(* IEC 61131-3 sources: mect_apps/TP1070_01_C/Monitoring/plc, 9 files *)

(* ---- Crosstable.gvl ---- *)
VAR_GLOBAL
	HeatingEnable AT %QX0.4.0:BOOL;
	HeatingSetPoint_A AT %QW0.8:INT;	(* piano sopra *)
	HeatingSetPoint_B AT %QW0.12:INT;	(* piano terra *)
	HeatingSetPoint_C AT %QW0.16:INT;	(* piano sotto *)
	HeatingDelta AT %QW0.20:INT;
	CoolingEnable AT %QX0.44.0:BOOL;
	CoolingSetPoint_A AT %QW0.48:INT;	(* piano sopra *)
	CoolingSetPoint_B AT %QW0.52:INT;	(* piano terra *)
	CoolingSetPoint_C AT %QW0.56:INT;	(* piano sotto *)
	SavedAlarmStatus AT %QW0.752:UINT;
	SavedAlarmConfig AT %QD0.756:UDINT;
	openvpn_restart_times AT %QD0.768:UDINT;
	is_PPP0_ON AT %QX0.772.0:BOOL;	(* isUP_ppp0() *)
	is_TUN0_ON AT %QX0.776.0:BOOL;	(* isUP_tun0() *)
	is_Caldaia_ON AT %QX0.780.0:BOOL;
	XX_Baudrate AT %IW0.804:UINT;	(* Baudrate MPNC005 device *)
	XX_NodeID AT %IW0.808:UINT;	(* Address MPNC005 device *)
	XX_HeartBeat AT %ID0.812:UDINT;	(* Life time MPNC005 device *)
	XX_AnInConf_A AT %QW0.816:UINT;	(* Analog inputs configuration MPNC030 module A *)
	XX_AnInConf_B AT %QW0.820:UINT;	(* Analog inputs configuration MPNC030 module B *)
	XX_AnInConf_C AT %QW0.824:UINT;	(* Analog inputs configuration MPNC030 module C *)
	XX_AnIn_A_1 AT %IW0.832:INT;	(* Analog input 1 value MPNC030 module A *)
	XX_AnIn_A_2 AT %IW0.836:INT;	(* Analog input 2 value MPNC030 module A *)
	XX_AnIn_A_3 AT %IW0.840:INT;	(* Analog input 3 value MPNC030 module A *)
	XX_AnIn_A_4 AT %IW0.844:INT;	(* Analog input 4 value MPNC030 module A *)
	XX_AnIn_B_1 AT %IW0.848:INT;	(* Analog input 1 value MPNC030 module B *)
	XX_AnIn_B_2 AT %IW0.852:INT;	(* Analog input 2 value MPNC030 module B *)
	XX_AnIn_B_3 AT %IW0.856:INT;	(* Analog input 3 value MPNC030 module B *)
	XX_AnIn_B_4 AT %IW0.860:INT;	(* Analog input 4 value MPNC030 module B *)
	XX_AnIn_C_1 AT %IW0.864:INT;	(* Analog input 1 value MPNC030 module C *)
	XX_AnIn_C_2 AT %IW0.868:INT;	(* Analog input 2 value MPNC030 module C *)
	XX_AnIn_C_3 AT %IW0.872:INT;	(* Analog input 3 value MPNC030 module C *)
	XX_AnIn_C_4 AT %IW0.876:INT;	(* Analog input 4 value MPNC030 module C *)
	XX_DigOut_A_1 AT %QX0.896.0:BOOL;	(* Digital output value bit 1 MPNC020 02 module A *)
	XX_DigOut_A_2 AT %QX0.900.0:BOOL;	(* Digital output value bit 2 MPNC020 02 module A *)
	XX_DigOut_A_3 AT %QX0.904.0:BOOL;	(* Digital output value bit 3 MPNC020 02 module A *)
	XX_DigOut_A_4 AT %QX0.908.0:BOOL;	(* Digital output value bit 4 MPNC020 02 module A *)
	XX_DigOut_A_5 AT %QX0.912.0:BOOL;	(* Digital output value bit 5 MPNC020 02 module A *)
	XX_DigOut_A_6 AT %QX0.916.0:BOOL;	(* Digital output value bit 6 MPNC020 02 module A *)
	XX_DigOut_A_7 AT %QX0.920.0:BOOL;	(* Digital output value bit 7 MPNC020 02 module A *)
	XX_DigOut_A_8 AT %QX0.924.0:BOOL;	(* Digital output value bit 8 MPNC020 02 module A *)
	XX_DigOut_A_9 AT %QX0.928.0:BOOL;	(* Digital output value bit 9 MPNC020 02 module A *)
	XX_DigOut_A_10 AT %QX0.932.0:BOOL;	(* Digital output value bit 10 MPNC020 02 module A *)
	XX_DigOut_A_11 AT %QX0.936.0:BOOL;	(* Digital output value bit 11 MPNC020 02 module A *)
	XX_DigOut_A_12 AT %QX0.940.0:BOOL;	(* Digital output value bit 12 MPNC020 02 module A *)
	XX_DigOut_A_13 AT %QX0.944.0:BOOL;	(* Digital output value bit 13 MPNC020 02 module A *)
	XX_DigOut_A_14 AT %QX0.948.0:BOOL;	(* Digital output value bit 14 MPNC020 02 module A *)
	XX_DigOut_A_15 AT %QX0.952.0:BOOL;	(* Digital output value bit 15 MPNC020 02 module A *)
	XX_DigOut_A_16 AT %QX0.956.0:BOOL;	(* Digital output value bit 16 MPNC020 02 module A *)
	XX_DigIn_A_1 AT %IX0.1152.0:BOOL;	(* Digital input value bit 1 MPNC020 01 module A *)
	XX_DigIn_A_2 AT %IX0.1156.0:BOOL;	(* Digital input value bit 2 MPNC020 01 module A *)
	XX_DigIn_A_3 AT %IX0.1160.0:BOOL;	(* Digital input value bit 3 MPNC020 01 module A *)
	XX_DigIn_A_4 AT %IX0.1164.0:BOOL;	(* Digital input value bit 4 MPNC020 01 module A *)
	XX_DigIn_A_5 AT %IX0.1168.0:BOOL;	(* Digital input value bit 5 MPNC020 01 module A *)
	XX_DigIn_A_6 AT %IX0.1172.0:BOOL;	(* Digital input value bit 6 MPNC020 01 module A *)
	XX_DigIn_A_7 AT %IX0.1176.0:BOOL;	(* Digital input value bit 7 MPNC020 01 module A *)
	XX_DigIn_A_8 AT %IX0.1180.0:BOOL;	(* Digital input value bit 8 MPNC020 01 module A *)
	XX_DigIn_A_9 AT %IX0.1184.0:BOOL;	(* Digital input value bit 9 MPNC020 01 module A *)
	XX_DigIn_A_10 AT %IX0.1188.0:BOOL;	(* Digital input value bit 10 MPNC020 01 module A *)
	XX_DigIn_A_11 AT %IX0.1192.0:BOOL;	(* Digital input value bit 11 MPNC020 01 module A *)
	XX_DigIn_A_12 AT %IX0.1196.0:BOOL;	(* Digital input value bit 12 MPNC020 01 module A *)
	XX_DigIn_A_13 AT %IX0.1200.0:BOOL;	(* Digital input value bit 13 MPNC020 01 module A *)
	XX_DigIn_A_14 AT %IX0.1204.0:BOOL;	(* Digital input value bit 14 MPNC020 01 module A *)
	XX_DigIn_A_15 AT %IX0.1208.0:BOOL;	(* Digital input value bit 15 MPNC020 01 module A *)
	XX_DigIn_A_16 AT %IX0.1212.0:BOOL;	(* Digital input value bit 16 MPNC020 01 module A *)
	XX_DigIn_B_1 AT %IX0.1216.0:BOOL;	(* Digital input value bit 1 MPNC020 01 module B *)
	XX_DigIn_B_2 AT %IX0.1220.0:BOOL;	(* Digital input value bit 2 MPNC020 01 module B *)
	XX_DigIn_B_3 AT %IX0.1224.0:BOOL;	(* Digital input value bit 3 MPNC020 01 module B *)
	XX_DigIn_B_4 AT %IX0.1228.0:BOOL;	(* Digital input value bit 4 MPNC020 01 module B *)
	XX_DigIn_B_5 AT %IX0.1232.0:BOOL;	(* Digital input value bit 5 MPNC020 01 module B *)
	XX_DigIn_B_6 AT %IX0.1236.0:BOOL;	(* Digital input value bit 6 MPNC020 01 module B *)
	XX_DigIn_B_7 AT %IX0.1240.0:BOOL;	(* Digital input value bit 7 MPNC020 01 module B *)
	XX_DigIn_B_8 AT %IX0.1244.0:BOOL;	(* Digital input value bit 8 MPNC020 01 module B *)
	XX_DigIn_B_9 AT %IX0.1248.0:BOOL;	(* Digital input value bit 9 MPNC020 01 module B *)
	XX_DigIn_B_10 AT %IX0.1252.0:BOOL;	(* Digital input value bit 10 MPNC020 01 module B *)
	XX_DigIn_B_11 AT %IX0.1256.0:BOOL;	(* Digital input value bit 11 MPNC020 01 module B *)
	XX_DigIn_B_12 AT %IX0.1260.0:BOOL;	(* Digital input value bit 12 MPNC020 01 module B *)
	XX_DigIn_B_13 AT %IX0.1264.0:BOOL;	(* Digital input value bit 13 MPNC020 01 module B *)
	XX_DigIn_B_14 AT %IX0.1268.0:BOOL;	(* Digital input value bit 14 MPNC020 01 module B *)
	XX_DigIn_B_15 AT %IX0.1272.0:BOOL;	(* Digital input value bit 15 MPNC020 01 module B *)
	XX_DigIn_B_16 AT %IX0.1276.0:BOOL;	(* Digital input value bit 16 MPNC020 01 module B *)
	XX_Reserved_1 AT %IW0.1408:UINT;
	XX_Reserved_2 AT %IW0.1412:UINT;
	XX_ColdJunctionT AT %IW0.1416:INT;	(* Cold junction temperature value *)
	XX_Reserved_3 AT %IW0.1420:UINT;
	XX_Reserved_4 AT %IW0.1424:UINT;
	XX_Reboot AT %QW0.1428:INT;	(* MPNC006 chain reboot *)
	XX_ModulesNumber AT %IW0.1432:UINT;	(* Number of modules *)
	XX_AnInConf_1 AT %QW0.1436:UINT;	(* Analog input 1 configuration MPNC005 *)
	XX_AnInConf_2 AT %QW0.1440:UINT;	(* Analog input 2 configuration MPNC005 *)
	XX_AnIn_1 AT %IW0.1444:INT;	(* Analog input 1 value MPNC005 *)
	XX_AnIn_2 AT %IW0.1448:INT;	(* Analog input 2 value MPNC005 *)
	XX_DigDir_1 AT %QX0.1452.0:BOOL;	(* Digital IO 1 configuration MPNC005 *)
	XX_DigDir_2 AT %QX0.1456.0:BOOL;	(* Digital IO 2 configuration MPNC005 *)
	XX_DigDir_3 AT %QX0.1460.0:BOOL;	(* Digital IO 3 configuration MPNC005 *)
	XX_DigDir_4 AT %QX0.1464.0:BOOL;	(* Digital IO 4 configuration MPNC005 *)
	XX_DigDir_5 AT %QX0.1468.0:BOOL;	(* Digital IO 5 configuration MPNC005 *)
	XX_DigDir_6 AT %QX0.1472.0:BOOL;	(* Digital IO 6 configuration MPNC005 *)
	XX_DigDir_7 AT %QX0.1476.0:BOOL;	(* Digital IO 7 configuration MPNC005 *)
	XX_DigDir_8 AT %QX0.1480.0:BOOL;	(* Digital IO 8 configuration MPNC005 *)
	XX_DigIn_1 AT %IX0.1484.0:BOOL;	(* Digital input 1 value MPNC005 *)
	XX_DigIn_2 AT %IX0.1488.0:BOOL;	(* Digital input 2 value MPNC005 *)
	XX_DigIn_3 AT %IX0.1492.0:BOOL;	(* Digital input 3 value MPNC005 *)
	XX_DigIn_4 AT %IX0.1496.0:BOOL;	(* Digital input 4 value MPNC005 *)
	XX_DigIn_5 AT %IX0.1500.0:BOOL;	(* Digital input 5 value MPNC005 *)
	XX_DigIn_6 AT %IX0.1504.0:BOOL;	(* Digital input 6 value MPNC005 *)
	XX_DigIn_7 AT %IX0.1508.0:BOOL;	(* Digital input 7 value MPNC005 *)
	XX_DigIn_8 AT %IX0.1512.0:BOOL;	(* Digital input 8 value MPNC005 *)
	XX_DigOut_1 AT %QX0.1516.0:BOOL;	(* Digital output 1 value MPNC005 *)
	XX_DigOut_2 AT %QX0.1520.0:BOOL;	(* Digital output 2 value MPNC005 *)
	XX_DigOut_3 AT %QX0.1524.0:BOOL;	(* Digital output 3 value MPNC005 *)
	XX_DigOut_4 AT %QX0.1528.0:BOOL;	(* Digital output 4 value MPNC005 *)
	XX_DigOut_5 AT %QX0.1532.0:BOOL;	(* Digital output 5 value MPNC005 *)
	XX_DigOut_6 AT %QX0.1536.0:BOOL;	(* Digital output 6 value MPNC005 *)
	XX_DigOut_7 AT %QX0.1540.0:BOOL;	(* Digital output 7 value MPNC005 *)
	XX_DigOut_8 AT %QX0.1544.0:BOOL;	(* Digital output 8 value MPNC005 *)
	XX_AnInFltr_1 AT %QW0.1548:UINT;	(* Analog input filter 1 MPNC006 *)
	XX_AnInFltr_2 AT %QW0.1552:UINT;	(* Analog input filter 2 MPNC006 *)
	XX_WatchDog AT %QW0.1556:UINT;	(* WatchDog Timer in Seconds *)
	XX_FirmwareVer AT %IW0.1644:UINT;	(* Firmware release MPNC006 *)
	XX_StatusWord AT %IW0.1648:UINT;	(* Status word MPNC006 *)
	SystemVoltage_0 AT %ID0.1656:REAL;	(* 0x0A 0x100C Tensione in V (PRINCIPALE) *)
	SysPowerFactor_0 AT %ID0.1660:REAL;	(* 0x0A 0x101E Fattore di Potenza 0 (PRINCIPALE) *)
	SysActivePower_0 AT %ID0.1664:REAL;	(* 0x0A 0x1026 Potenza Attiva 0 in W (PRINCIPALE) *)
	SysImpActiveEnergy_0 AT %ID0.1668:REAL;	(* 0x0A 0x1106 Energia Attiva Importata 0 in Wh (PRINCIPALE) *)
	SysExpActiveEnergy_0 AT %ID0.1672:REAL;	(* 0x0A 0x110E Energia Attiva Esportata 0 in Wh (PRINCIPALE) *)
	SysActivePower_1 AT %ID0.1676:REAL;	(* 0x0B 0x1026 Potenza Attiva 0 in W (FOTOVOLTAICO) *)
	SysImpActiveEnergy_1 AT %ID0.1680:REAL;	(* 0x0B 0x1106 Energia Attiva Importata 1 in Wh (FOTOVOLTAICO) *)
	SysExpActiveEnergy_1 AT %ID0.1684:REAL;	(* 0x0B 0x110E Energia Attiva Esportata 0 in Wh (FOTOVOLTAICO) *)
	SysActivePower_2 AT %ID0.1688:REAL;	(* 0x0C 0x1026 Potenza Attiva 0 in W (ESTERNI) *)
	SysImpActiveEnergy_2 AT %ID0.1692:REAL;	(* 0x0C 0x1106 Energia Attiva Importata 0 in Wh (ESTERNI) *)
	SysActivePower_3 AT %ID0.1696:REAL;	(* 0x0D 0x1026 Potenza Attiva 0 in W (PIANO SOPRA) *)
	SysImpActiveEnergy_3 AT %ID0.1700:REAL;	(* 0x0D 0x1106 Energia Attiva Importata 0 in Wh (PIANO SOPRA) *)
	SysActivePower_4 AT %ID0.1704:REAL;	(* 0x0E 0x1026 Potenza Attiva 0 in W (PIANO TERRA) *)
	SysImpActiveEnergy_4 AT %ID0.1708:REAL;	(* 0x0E 0x1106 Energia Attiva Importata 0 in Wh (PIANO TERRA) *)
	SysActivePower_5 AT %ID0.1712:REAL;	(* 0x0F 0x1026 Potenza Attiva 0 in W (PIANO SOTTO) *)
	SysImpActiveEnergy_5 AT %ID0.1716:REAL;	(* 0x0F 0x1106 Energia Attiva Importata 0 in Wh (PIANO SOTTO) *)
	SysActivePower_6 AT %ID0.1720:REAL;	(* 0x10 0x1026 Potenza Attiva 0 in W (AUTO ELETTRICA) *)
	SysImpActiveEnergy_6 AT %ID0.1724:REAL;	(* 0x10 0x1106 Energia Attiva Importata 0 in Wh (AUTO ELETTRICA) *)
	SysActivePower_7 AT %ID0.1728:REAL;	(* 0x11 0x1026 Potenza Attiva 0 in W (DEUMIDIFICATORE) *)
	SysImpActiveEnergy_7 AT %ID0.1732:REAL;	(* 0x11 0x1106 Energia Attiva Importata 0 in Wh (DEUMIDIFICATORE) *)
	SysActivePower_8 AT %ID0.1736:REAL;	(* 0x12 0x1026 Potenza Attiva 0 in W (LAVANDERIA) *)
	SysImpActiveEnergy_8 AT %ID0.1740:REAL;	(* 0x12 0x1106 Energia Attiva Importata 0 in Wh (LAVANDERIA) *)
	SysActivePower_9 AT %ID0.1744:REAL;	(* 0x13 0x1026 Potenza Attiva 0 in W (UPS) *)
	SysApparentPower_9 AT %ID0.1748:REAL;	(* 0x13 0x102E Potenza Apparente 0 in VA (UPS) *)
	SysImpActiveEnergy_9 AT %ID0.1752:REAL;	(* 0x13 0x1106 Energia Attiva Importata 0 in Wh (UPS) *)
	SysActivePower_10 AT %ID0.1756:REAL;	(* 0x14 0x1026 Potenza Attiva 0 in W (Puffer) *)
	SysImpActiveEnergy_10 AT %ID0.1760:REAL;	(* 0x14 0x1106 Energia Attiva Importata 0 in Wh (Puffer) *)
	SysActivePower_11 AT %QD0.1764:REAL;	(* 0x14 0x1026 Potenza Attiva 0 in W (Caldaia) *)
	SysImpActiveEnergy_11 AT %QD0.1768:REAL;	(* 0x14 0x1106 Energia Attiva Importata 0 in Wh (Caldaia) *)
	AlarmStatus AT %QW0.1996:UINT;
	Alarm AT %QX0.2000.0:BOOL;
	OK_DigIn_A_1 AT %QX0.2004.0:BOOL;
	OK_DigIn_A_2 AT %QX0.2008.0:BOOL;
	OK_DigIn_A_3 AT %QX0.2012.0:BOOL;
	OK_DigIn_A_4 AT %QX0.2016.0:BOOL;
	OK_DigIn_A_5 AT %QX0.2020.0:BOOL;
	OK_DigIn_A_6 AT %QX0.2024.0:BOOL;
	OK_DigIn_A_7 AT %QX0.2028.0:BOOL;
	OK_DigIn_A_8 AT %QX0.2032.0:BOOL;
	OK_DigIn_A_9 AT %QX0.2036.0:BOOL;
	OK_DigIn_A_10 AT %QX0.2040.0:BOOL;
	OK_DigIn_A_11 AT %QX0.2044.0:BOOL;
	OK_DigIn_A_12 AT %QX0.2048.0:BOOL;
	OK_DigIn_A_13 AT %QX0.2052.0:BOOL;
	OK_DigIn_A_14 AT %QX0.2056.0:BOOL;
	OK_DigIn_A_15 AT %QX0.2060.0:BOOL;
	OK_DigIn_A_16 AT %QX0.2064.0:BOOL;
	OK_DigIn_B_1 AT %QX0.2068.0:BOOL;
	OK_DigIn_B_2 AT %QX0.2072.0:BOOL;
	OK_DigIn_B_3 AT %QX0.2076.0:BOOL;
	OK_DigIn_B_4 AT %QX0.2080.0:BOOL;
	OK_DigIn_B_5 AT %QX0.2084.0:BOOL;
	OK_DigIn_B_6 AT %QX0.2088.0:BOOL;
	OK_DigIn_B_7 AT %QX0.2092.0:BOOL;
	OK_DigIn_B_8 AT %QX0.2096.0:BOOL;
	OK_DigIn_B_9 AT %QX0.2100.0:BOOL;
	OK_DigIn_B_10 AT %QX0.2104.0:BOOL;
	OK_DigIn_B_11 AT %QX0.2108.0:BOOL;
	OK_DigIn_B_12 AT %QX0.2112.0:BOOL;
	OK_DigIn_B_13 AT %QX0.2116.0:BOOL;
	OK_DigIn_B_14 AT %QX0.2120.0:BOOL;
	OK_DigIn_B_15 AT %QX0.2124.0:BOOL;
	OK_DigIn_B_16 AT %QX0.2128.0:BOOL;
	AlarmRising AT %IX0.2132.0:BOOL;
	AlarmArmed_A_1 AT %QX0.2404.0:BOOL;
	AlarmArmed_A_2 AT %QX0.2408.0:BOOL;
	AlarmArmed_A_3 AT %QX0.2412.0:BOOL;
	AlarmArmed_A_4 AT %QX0.2416.0:BOOL;
	AlarmArmed_A_5 AT %QX0.2420.0:BOOL;
	AlarmArmed_A_6 AT %QX0.2424.0:BOOL;
	AlarmArmed_A_7 AT %QX0.2428.0:BOOL;
	AlarmArmed_A_8 AT %QX0.2432.0:BOOL;
	AlarmArmed_A_9 AT %QX0.2436.0:BOOL;
	AlarmArmed_A_10 AT %QX0.2440.0:BOOL;
	AlarmArmed_A_11 AT %QX0.2444.0:BOOL;
	AlarmArmed_A_12 AT %QX0.2448.0:BOOL;
	AlarmArmed_A_13 AT %QX0.2452.0:BOOL;
	AlarmArmed_A_14 AT %QX0.2456.0:BOOL;
	AlarmArmed_A_15 AT %QX0.2460.0:BOOL;
	AlarmArmed_A_16 AT %QX0.2464.0:BOOL;
	AlarmArmed_B_1 AT %QX0.2468.0:BOOL;
	AlarmArmed_B_2 AT %QX0.2472.0:BOOL;
	AlarmArmed_B_3 AT %QX0.2476.0:BOOL;
	AlarmArmed_B_4 AT %QX0.2480.0:BOOL;
	AlarmArmed_B_5 AT %QX0.2484.0:BOOL;
	AlarmArmed_B_6 AT %QX0.2488.0:BOOL;
	AlarmArmed_B_7 AT %QX0.2492.0:BOOL;
	AlarmArmed_B_8 AT %QX0.2496.0:BOOL;
	AlarmArmed_B_9 AT %QX0.2500.0:BOOL;
	AlarmArmed_B_10 AT %QX0.2504.0:BOOL;
	AlarmArmed_B_11 AT %QX0.2508.0:BOOL;
	AlarmArmed_B_12 AT %QX0.2512.0:BOOL;
	AlarmArmed_B_13 AT %QX0.2516.0:BOOL;
	AlarmArmed_B_14 AT %QX0.2520.0:BOOL;
	AlarmArmed_B_15 AT %QX0.2524.0:BOOL;
	AlarmArmed_B_16 AT %QX0.2528.0:BOOL;
	TCP_is_Caldaia_ON AT %QX0.4000.0:BOOL;
	TCP_HeatingEnable AT %QX0.4004.0:BOOL;
	TCP_AnIn_A_1 AT %QW0.4008:INT;	(* Analog input 1 value MPNC030 module A *)
	TCP_AnIn_A_2 AT %QW0.4012:INT;	(* Analog input 2 value MPNC030 module A *)
	TCP_AnIn_A_3 AT %QW0.4016:INT;	(* Analog input 3 value MPNC030 module A *)
	TCP_AnIn_A_4 AT %QW0.4020:INT;	(* Analog input 4 value MPNC030 module A *)
	TCP_AnIn_B_1 AT %QW0.4024:INT;	(* Analog input 1 value MPNC030 module B *)
	TCP_AnIn_B_2 AT %QW0.4028:INT;	(* Analog input 2 value MPNC030 module B *)
	TCP_AnIn_B_3 AT %QW0.4032:INT;	(* Analog input 3 value MPNC030 module B *)
	TCP_AnIn_B_4 AT %QW0.4036:INT;	(* Analog input 4 value MPNC030 module B *)
	TCP_AnIn_C_1 AT %QW0.4040:INT;	(* Analog input 1 value MPNC030 module C *)
	TCP_AnIn_C_2 AT %QW0.4044:INT;	(* Analog input 2 value MPNC030 module C *)
	TCP_AnIn_C_3 AT %QW0.4048:INT;	(* Analog input 3 value MPNC030 module C *)
	TCP_AnIn_C_4 AT %QW0.4052:INT;	(* Analog input 3 value MPNC030 module C *)
	TCP_AnIn_1 AT %QW0.4056:INT;	(* Analog input 1 value MPNC005 *)
	TCP_AnIn_2 AT %QW0.4060:INT;	(* Analog input 2 value MPNC005 *)
	TCP_DigIn_1 AT %QX0.4064.0:BOOL;	(* Digital input 1 value MPNC005 *)
	TCP_DigIn_2 AT %QX0.4068.0:BOOL;	(* Digital input 2 value MPNC005 *)
	TCP_DigIn_3 AT %QX0.4072.0:BOOL;	(* Digital input 3 value MPNC005 *)
	TCP_DigIn_4 AT %QX0.4076.0:BOOL;	(* Digital input 4 value MPNC005 *)
	TCP_DigIn_5 AT %QX0.4080.0:BOOL;	(* Digital input 5 value MPNC005 *)
	TCP_DigIn_6 AT %QX0.4084.0:BOOL;	(* Digital input 6 value MPNC005 *)
	TCP_DigIn_7 AT %QX0.4088.0:BOOL;	(* Digital input 7 value MPNC005 *)
	TCP_DigIn_8 AT %QX0.4092.0:BOOL;	(* Digital input 8 value MPNC005 *)
	TCP_DigOut_1 AT %QX0.4096.0:BOOL;	(* Digital output 1 value MPNC005 *)
	TCP_DigOut_2 AT %QX0.4100.0:BOOL;	(* Digital output 2 value MPNC005 *)
	TCP_DigOut_3 AT %QX0.4104.0:BOOL;	(* Digital output 3 value MPNC005 *)
	TCP_DigOut_4 AT %QX0.4108.0:BOOL;	(* Digital output 4 value MPNC005 *)
	TCP_DigOut_5 AT %QX0.4112.0:BOOL;	(* Digital output 5 value MPNC005 *)
	TCP_DigOut_6 AT %QX0.4116.0:BOOL;	(* Digital output 6 value MPNC005 *)
	TCP_DigOut_7 AT %QX0.4120.0:BOOL;	(* Digital output 7 value MPNC005 *)
	TCP_DigOut_8 AT %QX0.4124.0:BOOL;	(* Digital output 8 value MPNC005 *)
	TCP_SystemVoltage_0 AT %QD0.4132:REAL;	(* 0x0A 0x100C Tensione in V (PRINCIPALE) *)
	TCP_SysPowerFactor_0 AT %QD0.4136:REAL;	(* 0x0A 0x101E Fattore di Potenza 0 (PRINCIPALE) *)
	TCP_SysActivePower_0 AT %QD0.4140:REAL;	(* 0x0A 0x1026 Potenza Attiva 0 in W (PRINCIPALE) *)
	TCP_SysImpActiveEnergy_0 AT %QD0.4144:REAL;	(* 0x0A 0x1106 Energia Attiva Importata 0 in Wh (PRINCIPALE) *)
	TCP_SysExpActiveEnergy_0 AT %QD0.4148:REAL;	(* 0x0A 0x110E Energia Attiva Esportata 0 in Wh (PRINCIPALE) *)
	TCP_SysActivePower_1 AT %QD0.4152:REAL;	(* 0x0B 0x1026 Potenza Attiva 0 in W (FOTOVOLTAICO) *)
	TCP_SysImpActiveEnergy_1 AT %QD0.4156:REAL;	(* 0x0B 0x1106 Energia Attiva Importata 1 in Wh (FOTOVOLTAICO) *)
	TCP_SysExpActiveEnergy_1 AT %QD0.4160:REAL;	(* 0x0B 0x110E Energia Attiva Esportata 0 in Wh (FOTOVOLTAICO) *)
	TCP_SysActivePower_2 AT %QD0.4164:REAL;	(* 0x0C 0x1026 Potenza Attiva 0 in W (ESTERNI) *)
	TCP_SysImpActiveEnergy_2 AT %QD0.4168:REAL;	(* 0x0C 0x1106 Energia Attiva Importata 0 in Wh (ESTERNI) *)
	TCP_SysActivePower_3 AT %QD0.4172:REAL;	(* 0x0D 0x1026 Potenza Attiva 0 in W (PIANO SOPRA) *)
	TCP_SysImpActiveEnergy_3 AT %QD0.4176:REAL;	(* 0x0D 0x1106 Energia Attiva Importata 0 in Wh (PIANO SOPRA) *)
	TCP_SysActivePower_4 AT %QD0.4180:REAL;	(* 0x0E 0x1026 Potenza Attiva 0 in W (PIANO TERRA) *)
	TCP_SysImpActiveEnergy_4 AT %QD0.4184:REAL;	(* 0x0E 0x1106 Energia Attiva Importata 0 in Wh (PIANO TERRA) *)
	TCP_SysActivePower_5 AT %QD0.4188:REAL;	(* 0x0F 0x1026 Potenza Attiva 0 in W (PIANO SOTTO) *)
	TCP_SysImpActiveEnergy_5 AT %QD0.4192:REAL;	(* 0x0F 0x1106 Energia Attiva Importata 0 in Wh (PIANO SOTTO) *)
	TCP_SysActivePower_6 AT %QD0.4196:REAL;	(* 0x10 0x1026 Potenza Attiva 0 in W (AUTO ELETTRICA) *)
	TCP_SysImpActiveEnergy_6 AT %QD0.4200:REAL;	(* 0x10 0x1106 Energia Attiva Importata 0 in Wh (AUTO ELETTRICA) *)
	TCP_SysActivePower_7 AT %QD0.4204:REAL;	(* 0x11 0x1026 Potenza Attiva 0 in W (DEUMIDIFICATORE) *)
	TCP_SysImpActiveEnergy_7 AT %QD0.4208:REAL;	(* 0x11 0x1106 Energia Attiva Importata 0 in Wh (DEUMIDIFICATORE) *)
	TCP_SysActivePower_8 AT %QD0.4212:REAL;	(* 0x12 0x1026 Potenza Attiva 0 in W (LAVANDERIA) *)
	TCP_SysImpActiveEnergy_8 AT %QD0.4216:REAL;	(* 0x12 0x1106 Energia Attiva Importata 0 in Wh (LAVANDERIA) *)
	TCP_SysActivePower_9 AT %QD0.4220:REAL;	(* 0x13 0x1026 Potenza Attiva 0 in W (UPS) *)
	TCP_SysApparentPower_9 AT %QD0.4224:REAL;	(* 0x13 0x102E Potenza Apparente 0 in VA (UPS) *)
	TCP_SysImpActiveEnergy_9 AT %QD0.4228:REAL;	(* 0x13 0x1106 Energia Attiva Importata 0 in Wh (UPS) *)
	TCP_SysActivePower_10 AT %QD0.4232:REAL;	(* 0x14 0x1026 Potenza Attiva 0 in W (Puffer) *)
	TCP_SysImpActiveEnergy_10 AT %QD0.4236:REAL;	(* 0x14 0x1106 Energia Attiva Importata 0 in Wh (Puffer) *)
	TCP_SysActivePower_11 AT %QD0.4240:REAL;	(* 0x14 0x1026 Potenza Attiva 0 in W (Caldaia) *)
	TCP_SysImpActiveEnergy_11 AT %QD0.4244:REAL;	(* 0x14 0x1106 Energia Attiva Importata 0 in Wh (Caldaia) *)
	TCP_Alarm AT %QX0.4252.0:BOOL;
	TCP_AlarmEnabled AT %QX0.4256.0:BOOL;
	TCP_AlarmArmed AT %QX0.4260.0:BOOL;
	TCP_DigOut_A_1 AT %QX0.4264.0:BOOL;	(* Digital output value bit 1 MPNC020 02 module A *)
	TCP_DigOut_A_2 AT %QX0.4268.0:BOOL;	(* Digital output value bit 2 MPNC020 02 module A *)
	TCP_DigOut_A_3 AT %QX0.4272.0:BOOL;	(* Digital output value bit 3 MPNC020 02 module A *)
	TCP_DigOut_A_4 AT %QX0.4276.0:BOOL;	(* Digital output value bit 4 MPNC020 02 module A *)
	TCP_DigOut_A_5 AT %QX0.4280.0:BOOL;	(* Digital output value bit 5 MPNC020 02 module A *)
	TCP_DigOut_A_6 AT %QX0.4284.0:BOOL;	(* Digital output value bit 6 MPNC020 02 module A *)
	TCP_DigOut_A_7 AT %QX0.4288.0:BOOL;	(* Digital output value bit 7 MPNC020 02 module A *)
	TCP_DigOut_A_8 AT %QX0.4292.0:BOOL;	(* Digital output value bit 8 MPNC020 02 module A *)
	TCP_DigOut_A_9 AT %QX0.4296.0:BOOL;	(* Digital output value bit 9 MPNC020 02 module A *)
	TCP_DigOut_A_10 AT %QX0.4300.0:BOOL;	(* Digital output value bit 10 MPNC020 02 module A *)
	TCP_DigOut_A_11 AT %QX0.4304.0:BOOL;	(* Digital output value bit 11 MPNC020 02 module A *)
	TCP_DigOut_A_12 AT %QX0.4308.0:BOOL;	(* Digital output value bit 12 MPNC020 02 module A *)
	TCP_DigOut_A_13 AT %QX0.4312.0:BOOL;	(* Digital output value bit 13 MPNC020 02 module A *)
	TCP_DigOut_A_14 AT %QX0.4316.0:BOOL;	(* Digital output value bit 14 MPNC020 02 module A *)
	TCP_DigOut_A_15 AT %QX0.4320.0:BOOL;	(* Digital output value bit 15 MPNC020 02 module A *)
	TCP_DigOut_A_16 AT %QX0.4324.0:BOOL;	(* Digital output value bit 16 MPNC020 02 module A *)
	TCP_DigIn_A_1 AT %QX0.4328.0:BOOL;	(* Digital input value bit 1 MPNC020 01 module A *)
	TCP_DigIn_A_2 AT %QX0.4332.0:BOOL;	(* Digital input value bit 2 MPNC020 01 module A *)
	TCP_DigIn_A_3 AT %QX0.4336.0:BOOL;	(* Digital input value bit 3 MPNC020 01 module A *)
	TCP_DigIn_A_4 AT %QX0.4340.0:BOOL;	(* Digital input value bit 4 MPNC020 01 module A *)
	TCP_DigIn_A_5 AT %QX0.4344.0:BOOL;	(* Digital input value bit 5 MPNC020 01 module A *)
	TCP_DigIn_A_6 AT %QX0.4348.0:BOOL;	(* Digital input value bit 6 MPNC020 01 module A *)
	TCP_DigIn_A_7 AT %QX0.4352.0:BOOL;	(* Digital input value bit 7 MPNC020 01 module A *)
	TCP_DigIn_A_8 AT %QX0.4356.0:BOOL;	(* Digital input value bit 8 MPNC020 01 module A *)
	TCP_DigIn_A_9 AT %QX0.4360.0:BOOL;	(* Digital input value bit 9 MPNC020 01 module A *)
	TCP_DigIn_A_10 AT %QX0.4364.0:BOOL;	(* Digital input value bit 10 MPNC020 01 module A *)
	TCP_DigIn_A_11 AT %QX0.4368.0:BOOL;	(* Digital input value bit 11 MPNC020 01 module A *)
	TCP_DigIn_A_12 AT %QX0.4372.0:BOOL;	(* Digital input value bit 12 MPNC020 01 module A *)
	TCP_DigIn_A_13 AT %QX0.4376.0:BOOL;	(* Digital input value bit 13 MPNC020 01 module A *)
	TCP_DigIn_A_14 AT %QX0.4380.0:BOOL;	(* Digital input value bit 14 MPNC020 01 module A *)
	TCP_DigIn_A_15 AT %QX0.4384.0:BOOL;	(* Digital input value bit 15 MPNC020 01 module A *)
	TCP_DigIn_A_16 AT %QX0.4388.0:BOOL;	(* Digital input value bit 16 MPNC020 01 module A *)
	TCP_DigIn_B_1 AT %QX0.4392.0:BOOL;	(* Digital input value bit 1 MPNC020 01 module B *)
	TCP_DigIn_B_2 AT %QX0.4396.0:BOOL;	(* Digital input value bit 2 MPNC020 01 module B *)
	TCP_DigIn_B_3 AT %QX0.4400.0:BOOL;	(* Digital input value bit 3 MPNC020 01 module B *)
	TCP_DigIn_B_4 AT %QX0.4404.0:BOOL;	(* Digital input value bit 4 MPNC020 01 module B *)
	TCP_DigIn_B_5 AT %QX0.4408.0:BOOL;	(* Digital input value bit 5 MPNC020 01 module B *)
	TCP_DigIn_B_6 AT %QX0.4412.0:BOOL;	(* Digital input value bit 6 MPNC020 01 module B *)
	TCP_DigIn_B_7 AT %QX0.4416.0:BOOL;	(* Digital input value bit 7 MPNC020 01 module B *)
	TCP_DigIn_B_8 AT %QX0.4420.0:BOOL;	(* Digital input value bit 8 MPNC020 01 module B *)
	TCP_DigIn_B_9 AT %QX0.4424.0:BOOL;	(* Digital input value bit 9 MPNC020 01 module B *)
	TCP_DigIn_B_10 AT %QX0.4428.0:BOOL;	(* Digital input value bit 10 MPNC020 01 module B *)
	TCP_DigIn_B_11 AT %QX0.4432.0:BOOL;	(* Digital input value bit 11 MPNC020 01 module B *)
	TCP_DigIn_B_12 AT %QX0.4436.0:BOOL;	(* Digital input value bit 12 MPNC020 01 module B *)
	TCP_DigIn_B_13 AT %QX0.4440.0:BOOL;	(* Digital input value bit 13 MPNC020 01 module B *)
	TCP_DigIn_B_14 AT %QX0.4444.0:BOOL;	(* Digital input value bit 14 MPNC020 01 module B *)
	TCP_DigIn_B_15 AT %QX0.4448.0:BOOL;	(* Digital input value bit 15 MPNC020 01 module B *)
	TCP_DigIn_B_16 AT %QX0.4452.0:BOOL;	(* Digital input value bit 16 MPNC020 01 module B *)
	TCP_OK_DigIn_A_1 AT %QX0.4460.0:BOOL;
	TCP_OK_DigIn_A_2 AT %QX0.4464.0:BOOL;
	TCP_OK_DigIn_A_3 AT %QX0.4468.0:BOOL;
	TCP_OK_DigIn_A_4 AT %QX0.4472.0:BOOL;
	TCP_OK_DigIn_A_5 AT %QX0.4476.0:BOOL;
	TCP_OK_DigIn_A_6 AT %QX0.4480.0:BOOL;
	TCP_OK_DigIn_A_7 AT %QX0.4484.0:BOOL;
	TCP_OK_DigIn_A_8 AT %QX0.4488.0:BOOL;
	TCP_OK_DigIn_A_9 AT %QX0.4492.0:BOOL;
	TCP_OK_DigIn_A_10 AT %QX0.4496.0:BOOL;
	TCP_OK_DigIn_A_11 AT %QX0.4500.0:BOOL;
	TCP_OK_DigIn_A_12 AT %QX0.4504.0:BOOL;
	TCP_OK_DigIn_A_13 AT %QX0.4508.0:BOOL;
	TCP_OK_DigIn_A_14 AT %QX0.4512.0:BOOL;
	TCP_OK_DigIn_A_15 AT %QX0.4516.0:BOOL;
	TCP_OK_DigIn_A_16 AT %QX0.4520.0:BOOL;
	TCP_OK_DigIn_B_1 AT %QX0.4524.0:BOOL;
	TCP_OK_DigIn_B_2 AT %QX0.4528.0:BOOL;
	TCP_OK_DigIn_B_3 AT %QX0.4532.0:BOOL;
	TCP_OK_DigIn_B_4 AT %QX0.4536.0:BOOL;
	TCP_OK_DigIn_B_5 AT %QX0.4540.0:BOOL;
	TCP_OK_DigIn_B_6 AT %QX0.4544.0:BOOL;
	TCP_OK_DigIn_B_7 AT %QX0.4548.0:BOOL;
	TCP_OK_DigIn_B_8 AT %QX0.4552.0:BOOL;
	TCP_OK_DigIn_B_9 AT %QX0.4556.0:BOOL;
	TCP_OK_DigIn_B_10 AT %QX0.4560.0:BOOL;
	TCP_OK_DigIn_B_11 AT %QX0.4564.0:BOOL;
	TCP_OK_DigIn_B_12 AT %QX0.4568.0:BOOL;
	TCP_OK_DigIn_B_13 AT %QX0.4572.0:BOOL;
	TCP_OK_DigIn_B_14 AT %QX0.4576.0:BOOL;
	TCP_OK_DigIn_B_15 AT %QX0.4580.0:BOOL;
	TCP_OK_DigIn_B_16 AT %QX0.4584.0:BOOL;
	TCP_AlarmStatus AT %QW0.4588:UINT;
	RTU0_TYPE_PORT AT %ID0.20000:UDINT;
	RTU0_BAUDRATE AT %ID0.20004:UDINT;
	RTU0_STATUS AT %ID0.20008:UDINT;
	RTU0_READS AT %ID0.20012:UDINT;
	RTU0_WRITES AT %ID0.20016:UDINT;
	RTU0_TIMEOUTS AT %ID0.20020:UDINT;
	RTU0_COMM_ERRORS AT %ID0.20024:UDINT;
	RTU0_LAST_ERROR AT %ID0.20028:UDINT;
	RTU0_WRITE_QUEUE AT %ID0.20032:UDINT;
	RTU0_BUS_LOAD AT %ID0.20036:UDINT;
	RTU1_TYPE_PORT AT %ID0.20040:UDINT;
	RTU1_BAUDRATE AT %ID0.20044:UDINT;
	RTU1_STATUS AT %ID0.20048:UDINT;
	RTU1_READS AT %ID0.20052:UDINT;
	RTU1_WRITES AT %ID0.20056:UDINT;
	RTU1_TIMEOUTS AT %ID0.20060:UDINT;
	RTU1_COMM_ERRORS AT %ID0.20064:UDINT;
	RTU1_LAST_ERROR AT %ID0.20068:UDINT;
	RTU1_WRITE_QUEUE AT %ID0.20072:UDINT;
	RTU1_BUS_LOAD AT %ID0.20076:UDINT;
	RTU3_TYPE_PORT AT %ID0.20080:UDINT;
	RTU3_BAUDRATE AT %ID0.20084:UDINT;
	RTU3_STATUS AT %ID0.20088:UDINT;
	RTU3_READS AT %ID0.20092:UDINT;
	RTU3_WRITES AT %ID0.20096:UDINT;
	RTU3_TIMEOUTS AT %ID0.20100:UDINT;
	RTU3_COMM_ERRORS AT %ID0.20104:UDINT;
	RTU3_LAST_ERROR AT %ID0.20108:UDINT;
	RTU3_WRITE_QUEUE AT %ID0.20112:UDINT;
	RTU3_BUS_LOAD AT %ID0.20116:UDINT;
	CAN0_TYPE_PORT AT %ID0.20120:UDINT;
	CAN0_BAUDRATE AT %ID0.20124:UDINT;
	CAN0_STATUS AT %ID0.20128:UDINT;
	CAN0_READS AT %ID0.20132:UDINT;
	CAN0_WRITES AT %ID0.20136:UDINT;
	CAN0_TIMEOUTS AT %ID0.20140:UDINT;
	CAN0_COMM_ERRORS AT %ID0.20144:UDINT;
	CAN0_LAST_ERROR AT %ID0.20148:UDINT;
	CAN0_WRITE_QUEUE AT %ID0.20152:UDINT;
	CAN0_BUS_LOAD AT %ID0.20156:UDINT;
	CAN1_TYPE_PORT AT %ID0.20160:UDINT;
	CAN1_BAUDRATE AT %ID0.20164:UDINT;
	CAN1_STATUS AT %ID0.20168:UDINT;
	CAN1_READS AT %ID0.20172:UDINT;
	CAN1_WRITES AT %ID0.20176:UDINT;
	CAN1_TIMEOUTS AT %ID0.20180:UDINT;
	CAN1_COMM_ERRORS AT %ID0.20184:UDINT;
	CAN1_LAST_ERROR AT %ID0.20188:UDINT;
	CAN1_WRITE_QUEUE AT %ID0.20192:UDINT;
	CAN1_BUS_LOAD AT %ID0.20196:UDINT;
	TCPS_TYPE_PORT AT %ID0.20200:UDINT;
	TCPS_IP_ADDRESS AT %ID0.20204:UDINT;
	TCPS_STATUS AT %ID0.20208:UDINT;
	TCPS_READS AT %ID0.20212:UDINT;
	TCPS_WRITES AT %ID0.20216:UDINT;
	TCPS_TIMEOUTS AT %ID0.20220:UDINT;
	TCPS_COMM_ERRORS AT %ID0.20224:UDINT;
	TCPS_LAST_ERROR AT %ID0.20228:UDINT;
	TCPS_WRITE_QUEUE AT %ID0.20232:UDINT;
	TCPS_BUS_LOAD AT %ID0.20236:UDINT;
	TCP0_TYPE_PORT AT %ID0.20240:UDINT;
	TCP0_IP_ADDRESS AT %ID0.20244:UDINT;
	TCP0_STATUS AT %ID0.20248:UDINT;
	TCP0_READS AT %ID0.20252:UDINT;
	TCP0_WRITES AT %ID0.20256:UDINT;
	TCP0_TIMEOUTS AT %ID0.20260:UDINT;
	TCP0_COMM_ERRORS AT %ID0.20264:UDINT;
	TCP0_LAST_ERROR AT %ID0.20268:UDINT;
	TCP0_WRITE_QUEUE AT %ID0.20272:UDINT;
	TCP0_BUS_LOAD AT %ID0.20276:UDINT;
	TCP1_TYPE_PORT AT %ID0.20280:UDINT;
	TCP1_IP_ADDRESS AT %ID0.20284:UDINT;
	TCP1_STATUS AT %ID0.20288:UDINT;
	TCP1_READS AT %ID0.20292:UDINT;
	TCP1_WRITES AT %ID0.20296:UDINT;
	TCP1_TIMEOUTS AT %ID0.20300:UDINT;
	TCP1_COMM_ERRORS AT %ID0.20304:UDINT;
	TCP1_LAST_ERROR AT %ID0.20308:UDINT;
	TCP1_WRITE_QUEUE AT %ID0.20312:UDINT;
	TCP1_BUS_LOAD AT %ID0.20316:UDINT;
	TCP2_TYPE_PORT AT %ID0.20320:UDINT;
	TCP2_IP_ADDRESS AT %ID0.20324:UDINT;
	TCP2_STATUS AT %ID0.20328:UDINT;
	TCP2_READS AT %ID0.20332:UDINT;
	TCP2_WRITES AT %ID0.20336:UDINT;
	TCP2_TIMEOUTS AT %ID0.20340:UDINT;
	TCP2_COMM_ERRORS AT %ID0.20344:UDINT;
	TCP2_LAST_ERROR AT %ID0.20348:UDINT;
	TCP2_WRITE_QUEUE AT %ID0.20352:UDINT;
	TCP2_BUS_LOAD AT %ID0.20356:UDINT;
	TCP3_TYPE_PORT AT %ID0.20360:UDINT;
	TCP3_IP_ADDRESS AT %ID0.20364:UDINT;
	TCP3_STATUS AT %ID0.20368:UDINT;
	TCP3_READS AT %ID0.20372:UDINT;
	TCP3_WRITES AT %ID0.20376:UDINT;
	TCP3_TIMEOUTS AT %ID0.20380:UDINT;
	TCP3_COMM_ERRORS AT %ID0.20384:UDINT;
	TCP3_LAST_ERROR AT %ID0.20388:UDINT;
	TCP3_WRITE_QUEUE AT %ID0.20392:UDINT;
	TCP3_BUS_LOAD AT %ID0.20396:UDINT;
	TCP4_TYPE_PORT AT %ID0.20400:UDINT;
	TCP4_IP_ADDRESS AT %ID0.20404:UDINT;
	TCP4_STATUS AT %ID0.20408:UDINT;
	TCP4_READS AT %ID0.20412:UDINT;
	TCP4_WRITES AT %ID0.20416:UDINT;
	TCP4_TIMEOUTS AT %ID0.20420:UDINT;
	TCP4_COMM_ERRORS AT %ID0.20424:UDINT;
	TCP4_LAST_ERROR AT %ID0.20428:UDINT;
	TCP4_WRITE_QUEUE AT %ID0.20432:UDINT;
	TCP4_BUS_LOAD AT %ID0.20436:UDINT;
	TCP5_TYPE_PORT AT %ID0.20440:UDINT;
	TCP5_IP_ADDRESS AT %ID0.20444:UDINT;
	TCP5_STATUS AT %ID0.20448:UDINT;
	TCP5_READS AT %ID0.20452:UDINT;
	TCP5_WRITES AT %ID0.20456:UDINT;
	TCP5_TIMEOUTS AT %ID0.20460:UDINT;
	TCP5_COMM_ERRORS AT %ID0.20464:UDINT;
	TCP5_LAST_ERROR AT %ID0.20468:UDINT;
	TCP5_WRITE_QUEUE AT %ID0.20472:UDINT;
	TCP5_BUS_LOAD AT %ID0.20476:UDINT;
	TCP6_TYPE_PORT AT %ID0.20480:UDINT;
	TCP6_IP_ADDRESS AT %ID0.20484:UDINT;
	TCP6_STATUS AT %ID0.20488:UDINT;
	TCP6_READS AT %ID0.20492:UDINT;
	TCP6_WRITES AT %ID0.20496:UDINT;
	TCP6_TIMEOUTS AT %ID0.20500:UDINT;
	TCP6_COMM_ERRORS AT %ID0.20504:UDINT;
	TCP6_LAST_ERROR AT %ID0.20508:UDINT;
	TCP6_WRITE_QUEUE AT %ID0.20512:UDINT;
	TCP6_BUS_LOAD AT %ID0.20516:UDINT;
	TCP7_TYPE_PORT AT %ID0.20520:UDINT;
	TCP7_IP_ADDRESS AT %ID0.20524:UDINT;
	TCP7_STATUS AT %ID0.20528:UDINT;
	TCP7_READS AT %ID0.20532:UDINT;
	TCP7_WRITES AT %ID0.20536:UDINT;
	TCP7_TIMEOUTS AT %ID0.20540:UDINT;
	TCP7_COMM_ERRORS AT %ID0.20544:UDINT;
	TCP7_LAST_ERROR AT %ID0.20548:UDINT;
	TCP7_WRITE_QUEUE AT %ID0.20552:UDINT;
	TCP7_BUS_LOAD AT %ID0.20556:UDINT;
	TCP8_TYPE_PORT AT %ID0.20560:UDINT;
	TCP8_IP_ADDRESS AT %ID0.20564:UDINT;
	TCP8_STATUS AT %ID0.20568:UDINT;
	TCP8_READS AT %ID0.20572:UDINT;
	TCP8_WRITES AT %ID0.20576:UDINT;
	TCP8_TIMEOUTS AT %ID0.20580:UDINT;
	TCP8_COMM_ERRORS AT %ID0.20584:UDINT;
	TCP8_LAST_ERROR AT %ID0.20588:UDINT;
	TCP8_WRITE_QUEUE AT %ID0.20592:UDINT;
	TCP8_BUS_LOAD AT %ID0.20596:UDINT;
	TCP9_TYPE_PORT AT %ID0.20600:UDINT;
	TCP9_IP_ADDRESS AT %ID0.20604:UDINT;
	TCP9_STATUS AT %ID0.20608:UDINT;
	TCP9_READS AT %ID0.20612:UDINT;
	TCP9_WRITES AT %ID0.20616:UDINT;
	TCP9_TIMEOUTS AT %ID0.20620:UDINT;
	TCP9_COMM_ERRORS AT %ID0.20624:UDINT;
	TCP9_LAST_ERROR AT %ID0.20628:UDINT;
	TCP9_WRITE_QUEUE AT %ID0.20632:UDINT;
	TCP9_BUS_LOAD AT %ID0.20636:UDINT;
	NODE_01_DEV_NODE AT %ID0.20688:UDINT;
	NODE_01_STATUS AT %ID0.20692:UDINT;
	NODE_02_DEV_NODE AT %ID0.20696:UDINT;
	NODE_02_STATUS AT %ID0.20700:UDINT;
	NODE_03_DEV_NODE AT %ID0.20704:UDINT;
	NODE_03_STATUS AT %ID0.20708:UDINT;
	NODE_04_DEV_NODE AT %ID0.20712:UDINT;
	NODE_04_STATUS AT %ID0.20716:UDINT;
	NODE_05_DEV_NODE AT %ID0.20720:UDINT;
	NODE_05_STATUS AT %ID0.20724:UDINT;
	NODE_06_DEV_NODE AT %ID0.20728:UDINT;
	NODE_06_STATUS AT %ID0.20732:UDINT;
	NODE_07_DEV_NODE AT %ID0.20736:UDINT;
	NODE_07_STATUS AT %ID0.20740:UDINT;
	NODE_08_DEV_NODE AT %ID0.20744:UDINT;
	NODE_08_STATUS AT %ID0.20748:UDINT;
	NODE_09_DEV_NODE AT %ID0.20752:UDINT;
	NODE_09_STATUS AT %ID0.20756:UDINT;
	NODE_10_DEV_NODE AT %ID0.20760:UDINT;
	NODE_10_STATUS AT %ID0.20764:UDINT;
	NODE_11_DEV_NODE AT %ID0.20768:UDINT;
	NODE_11_STATUS AT %ID0.20772:UDINT;
	NODE_12_DEV_NODE AT %ID0.20776:UDINT;
	NODE_12_STATUS AT %ID0.20780:UDINT;
	NODE_13_DEV_NODE AT %ID0.20784:UDINT;
	NODE_13_STATUS AT %ID0.20788:UDINT;
	NODE_14_DEV_NODE AT %ID0.20792:UDINT;
	NODE_14_STATUS AT %ID0.20796:UDINT;
	NODE_15_DEV_NODE AT %ID0.20800:UDINT;
	NODE_15_STATUS AT %ID0.20804:UDINT;
	NODE_16_DEV_NODE AT %ID0.20808:UDINT;
	NODE_16_STATUS AT %ID0.20812:UDINT;
	PLC_time AT %ID0.21560:REAL;	(* Seconds since boot (reset each 24h) *)
	PLC_timeMin AT %ID0.21564:REAL;	(* 10 seconds window start *)
	PLC_timeMax AT %ID0.21568:REAL;	(* 10 seconds window stop *)
	PLC_timeWin AT %QD0.21572:REAL;	(* Graph display window *)
	PLC_Version AT %IW0.21576:UINT;	(* Run Time version *)
	PLC_EngineStatus AT %IW0.21580:UINT;	(* PLC status *)
	PLC_ResetValues AT %QX0.21584.0:BOOL;	(* Diagnostic variables reset *)
	PLC_buzzerOn AT %QX0.21588.0:BOOL;	(* Buzzer sound (enable = 1 disable = 0) *)
	PLC_PLC_Version AT %QW0.21592:UINT;	(* PLC application version *)
	PLC_HMI_Version AT %QW0.21596:UINT;	(* HMI application version *)
	PLC_Year AT %IW0.21640:UINT;	(* Currently year *)
	PLC_Month AT %IW0.21644:UINT;	(* Currently month *)
	PLC_Day AT %IW0.21648:UINT;	(* Currently day *)
	PLC_Hours AT %IW0.21652:UINT;	(* Currently hour *)
	PLC_Minutes AT %IW0.21656:UINT;	(* Currently minutes *)
	PLC_Seconds AT %IW0.21660:UINT;	(* Currently seconds *)
	PLC_UPTIME_s AT %ID0.21664:UDINT;	(* Uptime in seconds (wraps in 136 years) *)
	PLC_UPTIME_cs AT %ID0.21668:UDINT;	(* Uptime in centiseconds = 10 ms (wraps in 497 days) *)
	PLC_WATCHDOGEN AT %QX0.21672.0:BOOL;	(* Enable Watchdog *)
	PLC_WATCHDOG_ms AT %QD0.21676:UDINT;	(* Reset Watchdog timer *)
	PLC_PRODUCT_ID AT %ID0.21680:UDINT;	(* TP/TPAC/TPLC Product ID (Hex) *)
	PLC_SERIAL_NUMBER AT %ID0.21684:UDINT;	(* TP/TPAC/TPLC Serial Number *)
	PLC_HMI_PAGE AT %QD0.21688:DINT;	(* HMI Page (page100=0x00000100) *)
	PLC_BEEP_VOLUME AT %QB0.21740:BYTE;	(* Beep volume (when buzzerOn) *)
	PLC_TOUCH_VOLUME AT %QB0.21744:BYTE;	(* Touch volume *)
	PLC_ALARM_VOLUME AT %QB0.21748:BYTE;	(* Alarm volume (when alarm) *)
	PLC_BUZZER AT %QD0.21752:UDINT;	(* Enable dynamic buzzer sound (0x44332211 up=0x11(%) on=0x22(cs) off=0x33(cs) rep=0x44(times)) *)
END_VAR

(* ---- RegolazioneOnOff.st ---- *)
(*[[
]]*)
FUNCTION RegolazioneOnOff
VAR_INPUT
    SetPoint : INT;
    Delta : INT;
    TheTemp : INT;
END_VAR
VAR_IN_OUT
    OnOff : BOOL;
END_VAR

	if TheTemp <= (SetPoint - Delta) then
		OnOff := true;
	elsif (SetPoint + Delta) < TheTemp then
		OnOff := false;
	else
		; (* OnOff rimane com'è *)
    end_if;

END_FUNCTION

(* ---- Alarms.st ---- *)
(*[[
]]*)
PROGRAM Alarms
#import "Crosstable.gvl"
#import "Resource1.gvl"

;

END_PROGRAM

(* ---- CheckDigIO.st ---- *)
(*[[
]]*)
PROGRAM CheckDigIO
#import "Crosstable.gvl"
#import "Resource1.gvl"

if (AlarmStatus = ALARM_STATUS_ZERO) then
    (* ... *)
	;

elsif (AlarmStatus = ALARM_STATUS_IDLE) then
	(* all ok *)

	OK_DigIn_A_1  := true; OK_DigIn_B_1  := true;
	OK_DigIn_A_2  := true; OK_DigIn_B_2  := true;
	OK_DigIn_A_3  := true; OK_DigIn_B_3  := true;
	OK_DigIn_A_4  := true; OK_DigIn_B_4  := true;
	OK_DigIn_A_5  := true; OK_DigIn_B_5  := true;
	OK_DigIn_A_6  := true; OK_DigIn_B_6  := true;
	OK_DigIn_A_7  := true; OK_DigIn_B_7  := true;
	OK_DigIn_A_8  := true; OK_DigIn_B_8  := true;
	OK_DigIn_A_9  := true; OK_DigIn_B_9  := true;
	OK_DigIn_A_10 := true; OK_DigIn_B_10 := true;
	OK_DigIn_A_11 := true; OK_DigIn_B_11 := true;
	OK_DigIn_A_12 := true; OK_DigIn_B_12 := true;
	OK_DigIn_A_13 := true; OK_DigIn_B_13 := true;
	OK_DigIn_A_14 := true; OK_DigIn_B_14 := true;
	OK_DigIn_A_15 := true; OK_DigIn_B_15 := true;
	OK_DigIn_A_16 := true; OK_DigIn_B_16 := true;

elsif (AlarmStatus = ALARM_STATUS_ARMED or AlarmStatus = ALARM_STATUS_ENABLED) then
	(* check DigIn, without memory *)

	OK_DigIn_A_1  := not AlarmArmed_A_1  or (XX_DigIn_A_1  = XX_DigOut_A_1 ); OK_DigIn_B_1  := not AlarmArmed_B_1  or (XX_DigIn_B_1  = XX_DigOut_A_1 );
	OK_DigIn_A_2  := not AlarmArmed_A_2  or (XX_DigIn_A_2  = XX_DigOut_A_2 ); OK_DigIn_B_2  := not AlarmArmed_B_2  or (XX_DigIn_B_2  = XX_DigOut_A_2 );
	OK_DigIn_A_3  := not AlarmArmed_A_3  or (XX_DigIn_A_3  = XX_DigOut_A_3 ); OK_DigIn_B_3  := not AlarmArmed_B_3  or (XX_DigIn_B_3  = XX_DigOut_A_3 );
	OK_DigIn_A_4  := not AlarmArmed_A_4  or (XX_DigIn_A_4  = XX_DigOut_A_4 ); OK_DigIn_B_4  := not AlarmArmed_B_4  or (XX_DigIn_B_4  = XX_DigOut_A_4 );
	OK_DigIn_A_5  := not AlarmArmed_A_5  or (XX_DigIn_A_5  = XX_DigOut_A_5 ); OK_DigIn_B_5  := not AlarmArmed_B_5  or (XX_DigIn_B_5  = XX_DigOut_A_5 );
	OK_DigIn_A_6  := not AlarmArmed_A_6  or (XX_DigIn_A_6  = XX_DigOut_A_6 ); OK_DigIn_B_6  := not AlarmArmed_B_6  or (XX_DigIn_B_6  = XX_DigOut_A_6 );
	OK_DigIn_A_7  := not AlarmArmed_A_7  or (XX_DigIn_A_7  = XX_DigOut_A_7 ); OK_DigIn_B_7  := not AlarmArmed_B_7  or (XX_DigIn_B_7  = XX_DigOut_A_7 );
	OK_DigIn_A_8  := not AlarmArmed_A_8  or (XX_DigIn_A_8  = XX_DigOut_A_8 ); OK_DigIn_B_8  := not AlarmArmed_B_8  or (XX_DigIn_B_8  = XX_DigOut_A_8 );
	OK_DigIn_A_9  := not AlarmArmed_A_9  or (XX_DigIn_A_9  = XX_DigOut_A_9 ); OK_DigIn_B_9  := not AlarmArmed_B_9  or (XX_DigIn_B_9  = XX_DigOut_A_9 );
	OK_DigIn_A_10 := not AlarmArmed_A_10 or (XX_DigIn_A_10 = XX_DigOut_A_10); OK_DigIn_B_10 := not AlarmArmed_B_10 or (XX_DigIn_B_10 = XX_DigOut_A_10);
	OK_DigIn_A_11 := not AlarmArmed_A_11 or (XX_DigIn_A_11 = XX_DigOut_A_11); OK_DigIn_B_11 := not AlarmArmed_B_11 or (XX_DigIn_B_11 = XX_DigOut_A_11);
	OK_DigIn_A_12 := not AlarmArmed_A_12 or (XX_DigIn_A_12 = XX_DigOut_A_12); OK_DigIn_B_12 := not AlarmArmed_B_12 or (XX_DigIn_B_12 = XX_DigOut_A_12);
	OK_DigIn_A_13 := not AlarmArmed_A_13 or (XX_DigIn_A_13 = XX_DigOut_A_13); OK_DigIn_B_13 := not AlarmArmed_B_13 or (XX_DigIn_B_13 = XX_DigOut_A_13);
	OK_DigIn_A_14 := not AlarmArmed_A_14 or (XX_DigIn_A_14 = XX_DigOut_A_14); OK_DigIn_B_14 := not AlarmArmed_B_14 or (XX_DigIn_B_14 = XX_DigOut_A_14);
	OK_DigIn_A_15 := not AlarmArmed_A_15 or (XX_DigIn_A_15 = XX_DigOut_A_15); OK_DigIn_B_15 := not AlarmArmed_B_15 or (XX_DigIn_B_15 = XX_DigOut_A_15);
	OK_DigIn_A_16 := not AlarmArmed_A_16 or (XX_DigIn_A_16 = XX_DigOut_A_16); OK_DigIn_B_16 := not AlarmArmed_B_16 or (XX_DigIn_B_16 = XX_DigOut_A_16);

elsif (AlarmStatus = ALARM_STATUS_RINGING or AlarmStatus = ALARM_STATUS_MUTED) then
	(* check DigIn, with memory *)

        OK_DigIn_A_1  := OK_DigIn_A_1  and (not AlarmArmed_A_1  or (XX_DigIn_A_1  = XX_DigOut_A_1 )); OK_DigIn_B_1  := OK_DigIn_B_1  and (not AlarmArmed_B_1  or (XX_DigIn_B_1  = XX_DigOut_A_1 ));
        OK_DigIn_A_2  := OK_DigIn_A_2  and (not AlarmArmed_A_2  or (XX_DigIn_A_2  = XX_DigOut_A_2 )); OK_DigIn_B_2  := OK_DigIn_B_2  and (not AlarmArmed_B_2  or (XX_DigIn_B_2  = XX_DigOut_A_2 ));
        OK_DigIn_A_3  := OK_DigIn_A_3  and (not AlarmArmed_A_3  or (XX_DigIn_A_3  = XX_DigOut_A_3 )); OK_DigIn_B_3  := OK_DigIn_B_3  and (not AlarmArmed_B_3  or (XX_DigIn_B_3  = XX_DigOut_A_3 ));
        OK_DigIn_A_4  := OK_DigIn_A_4  and (not AlarmArmed_A_4  or (XX_DigIn_A_4  = XX_DigOut_A_4 )); OK_DigIn_B_4  := OK_DigIn_B_4  and (not AlarmArmed_B_4  or (XX_DigIn_B_4  = XX_DigOut_A_4 ));
        OK_DigIn_A_5  := OK_DigIn_A_5  and (not AlarmArmed_A_5  or (XX_DigIn_A_5  = XX_DigOut_A_5 )); OK_DigIn_B_5  := OK_DigIn_B_5  and (not AlarmArmed_B_5  or (XX_DigIn_B_5  = XX_DigOut_A_5 ));
        OK_DigIn_A_6  := OK_DigIn_A_6  and (not AlarmArmed_A_6  or (XX_DigIn_A_6  = XX_DigOut_A_6 )); OK_DigIn_B_6  := OK_DigIn_B_6  and (not AlarmArmed_B_6  or (XX_DigIn_B_6  = XX_DigOut_A_6 ));
        OK_DigIn_A_7  := OK_DigIn_A_7  and (not AlarmArmed_A_7  or (XX_DigIn_A_7  = XX_DigOut_A_7 )); OK_DigIn_B_7  := OK_DigIn_B_7  and (not AlarmArmed_B_7  or (XX_DigIn_B_7  = XX_DigOut_A_7 ));
        OK_DigIn_A_8  := OK_DigIn_A_8  and (not AlarmArmed_A_8  or (XX_DigIn_A_8  = XX_DigOut_A_8 )); OK_DigIn_B_8  := OK_DigIn_B_8  and (not AlarmArmed_B_8  or (XX_DigIn_B_8  = XX_DigOut_A_8 ));
        OK_DigIn_A_9  := OK_DigIn_A_9  and (not AlarmArmed_A_9  or (XX_DigIn_A_9  = XX_DigOut_A_9 )); OK_DigIn_B_9  := OK_DigIn_B_9  and (not AlarmArmed_B_9  or (XX_DigIn_B_9  = XX_DigOut_A_9 ));
        OK_DigIn_A_10 := OK_DigIn_A_10 and (not AlarmArmed_A_10 or (XX_DigIn_A_10 = XX_DigOut_A_10)); OK_DigIn_B_10 := OK_DigIn_B_10 and (not AlarmArmed_B_10 or (XX_DigIn_B_10 = XX_DigOut_A_10));
        OK_DigIn_A_11 := OK_DigIn_A_11 and (not AlarmArmed_A_11 or (XX_DigIn_A_11 = XX_DigOut_A_11)); OK_DigIn_B_11 := OK_DigIn_B_11 and (not AlarmArmed_B_11 or (XX_DigIn_B_11 = XX_DigOut_A_11));
        OK_DigIn_A_12 := OK_DigIn_A_12 and (not AlarmArmed_A_12 or (XX_DigIn_A_12 = XX_DigOut_A_12)); OK_DigIn_B_12 := OK_DigIn_B_12 and (not AlarmArmed_B_12 or (XX_DigIn_B_12 = XX_DigOut_A_12));
        OK_DigIn_A_13 := OK_DigIn_A_13 and (not AlarmArmed_A_13 or (XX_DigIn_A_13 = XX_DigOut_A_13)); OK_DigIn_B_13 := OK_DigIn_B_13 and (not AlarmArmed_B_13 or (XX_DigIn_B_13 = XX_DigOut_A_13));
        OK_DigIn_A_14 := OK_DigIn_A_14 and (not AlarmArmed_A_14 or (XX_DigIn_A_14 = XX_DigOut_A_14)); OK_DigIn_B_14 := OK_DigIn_B_14 and (not AlarmArmed_B_14 or (XX_DigIn_B_14 = XX_DigOut_A_14));
        OK_DigIn_A_15 := OK_DigIn_A_15 and (not AlarmArmed_A_15 or (XX_DigIn_A_15 = XX_DigOut_A_15)); OK_DigIn_B_15 := OK_DigIn_B_15 and (not AlarmArmed_B_15 or (XX_DigIn_B_15 = XX_DigOut_A_15));
        OK_DigIn_A_16 := OK_DigIn_A_16 and (not AlarmArmed_A_16 or (XX_DigIn_A_16 = XX_DigOut_A_16)); OK_DigIn_B_16 := OK_DigIn_B_16 and (not AlarmArmed_B_16 or (XX_DigIn_B_16 = XX_DigOut_A_16));

else
	;

end_if;

END_PROGRAM

(* ---- CheckOK.st ---- *)
(*[[
]]*)
PROGRAM CheckOK
#import "Crosstable.gvl"
#import "Resource1.gvl"

case AlarmStatus of
	ALARM_STATUS_ZERO    :
		Alarm := false;
		(* AlarmStatus changed by hmi/page300  *)
	ALARM_STATUS_IDLE    :
		Alarm := false;
		(* AlarmStatus changed by hmi/page300 *)
	ALARM_STATUS_ARMED   :
		Alarm := false;
		(* AlarmStatus changed by hmi/page300 *)
	ALARM_STATUS_ENABLED :
		if ( OK_DigIn_A_1  and OK_DigIn_B_1  and
			 OK_DigIn_A_2  and OK_DigIn_B_2  and
			 OK_DigIn_A_3  and OK_DigIn_B_3  and
			 OK_DigIn_A_4  and OK_DigIn_B_4  and
			 OK_DigIn_A_5  and OK_DigIn_B_5  and
			 OK_DigIn_A_6  and OK_DigIn_B_6  and
			 OK_DigIn_A_7  and OK_DigIn_B_7  and
			 OK_DigIn_A_8  and OK_DigIn_B_8  and
			 OK_DigIn_A_9  and OK_DigIn_B_9  and
			 OK_DigIn_A_10 and OK_DigIn_B_10 and
			 OK_DigIn_A_11 and OK_DigIn_B_11 and
			 OK_DigIn_A_12 and OK_DigIn_B_12 and
			 OK_DigIn_A_13 and OK_DigIn_B_13 and
			 OK_DigIn_A_14 and OK_DigIn_B_14 and
			 OK_DigIn_A_15 and OK_DigIn_B_15 and
			 OK_DigIn_A_16 and OK_DigIn_B_16 ) then
			Alarm := false; (* all ok, *)
			(* AlarmStatus changed by hmi/page300 *)
		else
			Alarm := true;
			AlarmStatus := ALARM_STATUS_RINGING;
			SavedAlarmStatus := ALARM_STATUS_RINGING;
		end_if;
	ALARM_STATUS_RINGING :
		Alarm := true; (* persistent *)
		(* AlarmStatus changed by hmi/page300 *)
	ALARM_STATUS_MUTED   :
		Alarm := true; (* persistent *)
		(* AlarmStatus changed by hmi/page300 *)
else
	;
end_case;

END_PROGRAM

(* ---- Init.st ---- *)
(*[[
]]*)
PROGRAM Init
#import "Crosstable.gvl"
#import "Resource1.gvl"

	AlarmStatus := ALARM_STATUS_ZERO; (* vedi hmi/page300 *)
	XX_WatchDog := 1; (* MPNC DigOut watchdog 1 s (see also hmi/automation.cpp:setup() *)

END_PROGRAM

(* ---- Normal.st ---- *)
(*[[
]]*)
PROGRAM Normal
#import "Crosstable.gvl"
#import "Resource1.gvl"
VAR

END_VAR

	is_Caldaia_ON := XX_DigIn_6 or XX_DigIn_7 or XX_DigIn_8;

END_PROGRAM

(* ---- Slow.st ---- *)
(*[[
]]*)
PROGRAM Slow
#import "Crosstable.gvl"
#import "Resource1.gvl"
VAR
	ActivePower : REAL;
	OtherPowers : REAL;
END_VAR

	ActivePower := SysActivePower_0 (* PRINCIPALE     *) + SysActivePower_1 (* FOTOVOLTAICO    *);

	OtherPowers := SysActivePower_2 (* ESTERNI        *) + SysActivePower_3 (* PIANO SOPRA     *)
				 + SysActivePower_4 (* PIANO TERRA    *) + SysActivePower_5 (* PIANO SOTTO     *)
				 + SysActivePower_6 (* AUTO ELETTRICA *) + SysActivePower_7 (* DEUMIDIFICATORE *)
				 + SysActivePower_8 (* LAVANDERIA     *) + SysActivePower_9 (* UPS             *)
				 + SysActivePower_10(* PUFFER         *)                                         ;

	SysActivePower_11 (* CALDAIA *) := ActivePower - OtherPowers;

	(*******************************************************************************************)

	TCP_is_Caldaia_ON          := is_Caldaia_ON        ;
    TCP_HeatingEnable          := HeatingEnable        ;

	TCP_AnIn_A_1               := XX_AnIn_A_1          ;
	TCP_AnIn_A_2               := XX_AnIn_A_2          ;
	TCP_AnIn_A_3               := XX_AnIn_A_3          ;
	TCP_AnIn_A_4               := XX_AnIn_A_4          ;
	TCP_AnIn_B_1               := XX_AnIn_B_1          ;
	TCP_AnIn_B_2               := XX_AnIn_B_2          ;
	TCP_AnIn_B_3               := XX_AnIn_B_3          ;
	TCP_AnIn_B_4               := XX_AnIn_B_4          ;
	TCP_AnIn_C_1               := XX_AnIn_C_1          ;
	TCP_AnIn_C_2               := XX_AnIn_C_2          ;
	TCP_AnIn_C_3               := XX_AnIn_C_3          ;
	TCP_AnIn_C_4               := XX_AnIn_C_4          ;
	TCP_AnIn_1                 := XX_AnIn_1            ;
	TCP_AnIn_2                 := XX_AnIn_2            ;
	TCP_DigIn_1                := XX_DigIn_1           ;
	TCP_DigIn_2                := XX_DigIn_2           ;
	TCP_DigIn_3                := XX_DigIn_3           ;
	TCP_DigIn_4                := XX_DigIn_4           ;
	TCP_DigIn_5                := XX_DigIn_5           ;
	TCP_DigIn_6                := XX_DigIn_6           ;
	TCP_DigIn_7                := XX_DigIn_7           ;
	TCP_DigIn_8                := XX_DigIn_8           ;
	TCP_DigOut_1               := XX_DigOut_1          ;
	TCP_DigOut_2               := XX_DigOut_2          ;
	TCP_DigOut_3               := XX_DigOut_3          ;
	TCP_DigOut_4               := XX_DigOut_4          ;
	TCP_DigOut_5               := XX_DigOut_5          ;
	TCP_DigOut_6               := XX_DigOut_6          ;
	TCP_DigOut_7               := XX_DigOut_7          ;
	TCP_DigOut_8               := XX_DigOut_8          ;
	                                                   ;
	TCP_SystemVoltage_0        := SystemVoltage_0      ;
	TCP_SysPowerFactor_0       := SysPowerFactor_0     ;
	TCP_SysActivePower_0       := SysActivePower_0     ;
	TCP_SysImpActiveEnergy_0   := SysImpActiveEnergy_0 ;
	TCP_SysExpActiveEnergy_0   := SysExpActiveEnergy_0 ;
	TCP_SysActivePower_1       := SysActivePower_1     ;
	TCP_SysImpActiveEnergy_1   := SysImpActiveEnergy_1 ;
	TCP_SysExpActiveEnergy_1   := SysExpActiveEnergy_1 ;
	TCP_SysActivePower_2       := SysActivePower_2     ;
	TCP_SysImpActiveEnergy_2   := SysImpActiveEnergy_2 ;
	TCP_SysActivePower_3       := SysActivePower_3     ;
	TCP_SysImpActiveEnergy_3   := SysImpActiveEnergy_3 ;
	TCP_SysActivePower_4       := SysActivePower_4     ;
	TCP_SysImpActiveEnergy_4   := SysImpActiveEnergy_4 ;
	TCP_SysActivePower_5       := SysActivePower_5     ;
	TCP_SysImpActiveEnergy_5   := SysImpActiveEnergy_5 ;
	TCP_SysActivePower_6       := SysActivePower_6     ;
	TCP_SysImpActiveEnergy_6   := SysImpActiveEnergy_6 ;
	TCP_SysActivePower_7       := SysActivePower_7     ;
	TCP_SysImpActiveEnergy_7   := SysImpActiveEnergy_7 ;
	TCP_SysActivePower_8       := SysActivePower_8     ;
	TCP_SysImpActiveEnergy_8   := SysImpActiveEnergy_8 ;
	TCP_SysActivePower_9       := SysActivePower_9     ;
	TCP_SysApparentPower_9     := SysApparentPower_9   ;
	TCP_SysImpActiveEnergy_9   := SysImpActiveEnergy_9 ;
	TCP_SysActivePower_10      := SysActivePower_10    ;
	TCP_SysImpActiveEnergy_10  := SysImpActiveEnergy_10;
	TCP_SysActivePower_11      := SysActivePower_11    ;
	TCP_SysImpActiveEnergy_11  := SysImpActiveEnergy_11;

    TCP_Alarm		 := Alarm		 ;
	case AlarmStatus of
		ALARM_STATUS_ZERO:    TCP_AlarmEnabled := false; TCP_AlarmArmed := false;
		ALARM_STATUS_IDLE:    TCP_AlarmEnabled := false; TCP_AlarmArmed := false;
		ALARM_STATUS_ARMED:   TCP_AlarmEnabled := false; TCP_AlarmArmed := true;
  		ALARM_STATUS_ENABLED: TCP_AlarmEnabled := true;  TCP_AlarmArmed := true;
  		ALARM_STATUS_RINGING: TCP_AlarmEnabled := true;  TCP_AlarmArmed := true;
  		ALARM_STATUS_MUTED:   TCP_AlarmEnabled := false; TCP_AlarmArmed := true;
	else
		;
    end_case;

    TCP_DigOut_A_1  :=  XX_DigOut_A_1  ;
    TCP_DigOut_A_2  :=  XX_DigOut_A_2  ;
    TCP_DigOut_A_3  :=  XX_DigOut_A_3  ;
    TCP_DigOut_A_4  :=  XX_DigOut_A_4  ;
    TCP_DigOut_A_5  :=  XX_DigOut_A_5  ;
    TCP_DigOut_A_6  :=  XX_DigOut_A_6  ;
    TCP_DigOut_A_7  :=  XX_DigOut_A_7  ;
    TCP_DigOut_A_8  :=  XX_DigOut_A_8  ;
    TCP_DigOut_A_9  :=  XX_DigOut_A_9  ;
    TCP_DigOut_A_10 :=  XX_DigOut_A_10 ;
    TCP_DigOut_A_11 :=  XX_DigOut_A_11 ;
    TCP_DigOut_A_12 :=  XX_DigOut_A_12 ;
    TCP_DigOut_A_13 :=  XX_DigOut_A_13 ;
    TCP_DigOut_A_14 :=  XX_DigOut_A_14 ;
    TCP_DigOut_A_15 :=  XX_DigOut_A_15 ;
    TCP_DigOut_A_16 :=  XX_DigOut_A_16 ;

    TCP_DigIn_A_1   :=  XX_DigIn_A_1   ;
    TCP_DigIn_A_2   :=  XX_DigIn_A_2   ;
    TCP_DigIn_A_3   :=  XX_DigIn_A_3   ;
    TCP_DigIn_A_4   :=  XX_DigIn_A_4   ;
    TCP_DigIn_A_5   :=  XX_DigIn_A_5   ;
    TCP_DigIn_A_6   :=  XX_DigIn_A_6   ;
    TCP_DigIn_A_7   :=  XX_DigIn_A_7   ;
    TCP_DigIn_A_8   :=  XX_DigIn_A_8   ;
    TCP_DigIn_A_9   :=  XX_DigIn_A_9   ;
    TCP_DigIn_A_10  :=  XX_DigIn_A_10  ;
    TCP_DigIn_A_11  :=  XX_DigIn_A_11  ;
    TCP_DigIn_A_12  :=  XX_DigIn_A_12  ;
    TCP_DigIn_A_13  :=  XX_DigIn_A_13  ;
    TCP_DigIn_A_14  :=  XX_DigIn_A_14  ;
    TCP_DigIn_A_15  :=  XX_DigIn_A_15  ;
    TCP_DigIn_A_16  :=  XX_DigIn_A_16  ;
    TCP_DigIn_B_1   :=  XX_DigIn_B_1   ;
    TCP_DigIn_B_2   :=  XX_DigIn_B_2   ;
    TCP_DigIn_B_3   :=  XX_DigIn_B_3   ;
    TCP_DigIn_B_4   :=  XX_DigIn_B_4   ;
    TCP_DigIn_B_5   :=  XX_DigIn_B_5   ;
    TCP_DigIn_B_6   :=  XX_DigIn_B_6   ;
    TCP_DigIn_B_7   :=  XX_DigIn_B_7   ;
    TCP_DigIn_B_8   :=  XX_DigIn_B_8   ;
    TCP_DigIn_B_9   :=  XX_DigIn_B_9   ;
    TCP_DigIn_B_10  :=  XX_DigIn_B_10  ;
    TCP_DigIn_B_11  :=  XX_DigIn_B_11  ;
    TCP_DigIn_B_12  :=  XX_DigIn_B_12  ;
    TCP_DigIn_B_13  :=  XX_DigIn_B_13  ;
    TCP_DigIn_B_14  :=  XX_DigIn_B_14  ;
    TCP_DigIn_B_15  :=  XX_DigIn_B_15  ;
    TCP_DigIn_B_16  :=  XX_DigIn_B_16  ;

    TCP_OK_DigIn_A_1  := OK_DigIn_A_1  ;
    TCP_OK_DigIn_A_2  := OK_DigIn_A_2  ;
    TCP_OK_DigIn_A_3  := OK_DigIn_A_3  ;
    TCP_OK_DigIn_A_4  := OK_DigIn_A_4  ;
    TCP_OK_DigIn_A_5  := OK_DigIn_A_5  ;
    TCP_OK_DigIn_A_6  := OK_DigIn_A_6  ;
    TCP_OK_DigIn_A_7  := OK_DigIn_A_7  ;
    TCP_OK_DigIn_A_8  := OK_DigIn_A_8  ;
    TCP_OK_DigIn_A_9  := OK_DigIn_A_9  ;
    TCP_OK_DigIn_A_10 := OK_DigIn_A_10 ;
    TCP_OK_DigIn_A_11 := OK_DigIn_A_11 ;
    TCP_OK_DigIn_A_12 := OK_DigIn_A_12 ;
    TCP_OK_DigIn_A_13 := OK_DigIn_A_13 ;
    TCP_OK_DigIn_A_14 := OK_DigIn_A_14 ;
    TCP_OK_DigIn_A_15 := OK_DigIn_A_15 ;
    TCP_OK_DigIn_A_16 := OK_DigIn_A_16 ;
    TCP_OK_DigIn_B_1  := OK_DigIn_B_1  ;
    TCP_OK_DigIn_B_2  := OK_DigIn_B_2  ;
    TCP_OK_DigIn_B_3  := OK_DigIn_B_3  ;
    TCP_OK_DigIn_B_4  := OK_DigIn_B_4  ;
    TCP_OK_DigIn_B_5  := OK_DigIn_B_5  ;
    TCP_OK_DigIn_B_6  := OK_DigIn_B_6  ;
    TCP_OK_DigIn_B_7  := OK_DigIn_B_7  ;
    TCP_OK_DigIn_B_8  := OK_DigIn_B_8  ;
    TCP_OK_DigIn_B_9  := OK_DigIn_B_9  ;
    TCP_OK_DigIn_B_10 := OK_DigIn_B_10 ;
    TCP_OK_DigIn_B_11 := OK_DigIn_B_11 ;
    TCP_OK_DigIn_B_12 := OK_DigIn_B_12 ;
    TCP_OK_DigIn_B_13 := OK_DigIn_B_13 ;
    TCP_OK_DigIn_B_14 := OK_DigIn_B_14 ;
    TCP_OK_DigIn_B_15 := OK_DigIn_B_15 ;
    TCP_OK_DigIn_B_16 := OK_DigIn_B_16 ;

	TCP_AlarmStatus := AlarmStatus;

END_PROGRAM

(* ---- VerySlow.st ---- *)
(*[[
]]*)
PROGRAM VerySlow
#import "Crosstable.gvl"
#import "Resource1.gvl"
VAR
END_VAR

	if (XX_AnIn_A_4 < 50) then
		(* transitorio all'accensione *)
		MPT91_Set_point := 50; (* 5.0 °C *)
	else
		(* l'acqua nel puffer, per essere utile, deve essere più calda di quella nei termosifoni *)
		MPT91_Set_point := XX_AnIn_A_4 + 10; (* T_ritorno + 1.0 °C *)
	end_if;

END_PROGRAM
